PROGRAM PRG_05_Carriage
VAR
	R_TRIG_0: R_TRIG;
	R_TRIG_2: R_TRIG;
	bCarriageRt: BOOL;
	bCarriageLt: BOOL;
	lCarriageLeftLimit: LREAL;
	lCarriageRightLimit: LREAL;
	RS_CarriageCentre: RS;
	
	TOF_CarriageEN: TOF;
	R_TRIG_1: R_TRIG;
END_VAR

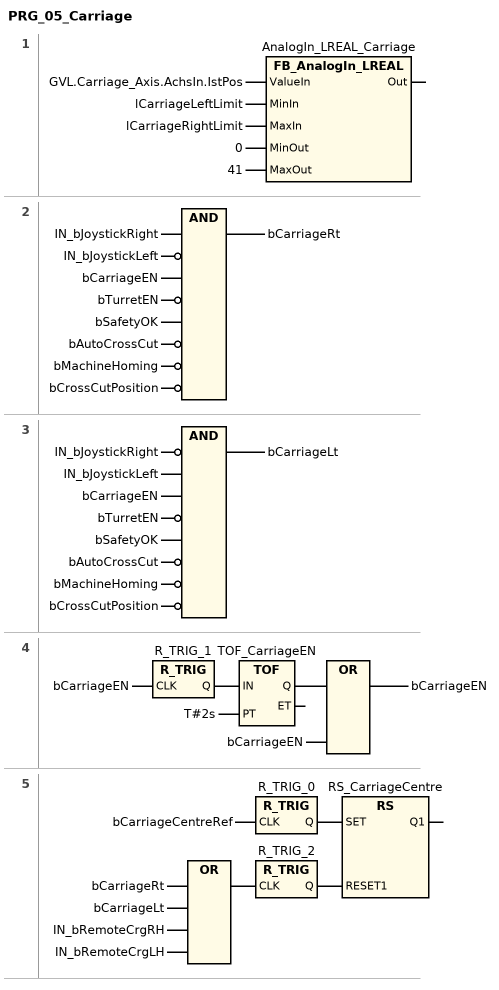
// NETWORK 1
AnalogIn_LREAL_Carriage(
    ValueIn := GVL.Carriage_Axis.AchsIn.IstPos,
    MinIn := lCarriageLeftLimit,
    MaxIn := lCarriageRightLimit,
    MinOut := 0,
    MaxOut := 41); // FB_AnalogIn_LREAL

// NETWORK 2
bCarriageRt := IN_bJoystickRight AND NOT IN_bJoystickLeft AND bCarriageEN AND NOT bTurretEN AND bSafetyOK AND NOT bAutoCrossCut AND NOT bMachineHoming AND NOT bCrossCutPosition;

// NETWORK 3
bCarriageLt := NOT IN_bJoystickRight AND IN_bJoystickLeft AND bCarriageEN AND NOT bTurretEN AND bSafetyOK AND NOT bAutoCrossCut AND NOT bMachineHoming AND NOT bCrossCutPosition;

// NETWORK 4
R_TRIG_1(CLK := bCarriageEN); // R_TRIG
TOF_CarriageEN(IN := R_TRIG_1.Q, PT := T#2s); // TOF
bCarriageEN := TOF_CarriageEN.Q OR bCarriageEN;

// NETWORK 5
R_TRIG_0(CLK := bCarriageCentreRef); // R_TRIG
R_TRIG_2(CLK := bCarriageRt OR bCarriageLt OR IN_bRemoteCrgRH OR IN_bRemoteCrgLH); // R_TRIG
RS_CarriageCentre(SET := R_TRIG_0.Q, RESET1 := R_TRIG_2.Q); // RS

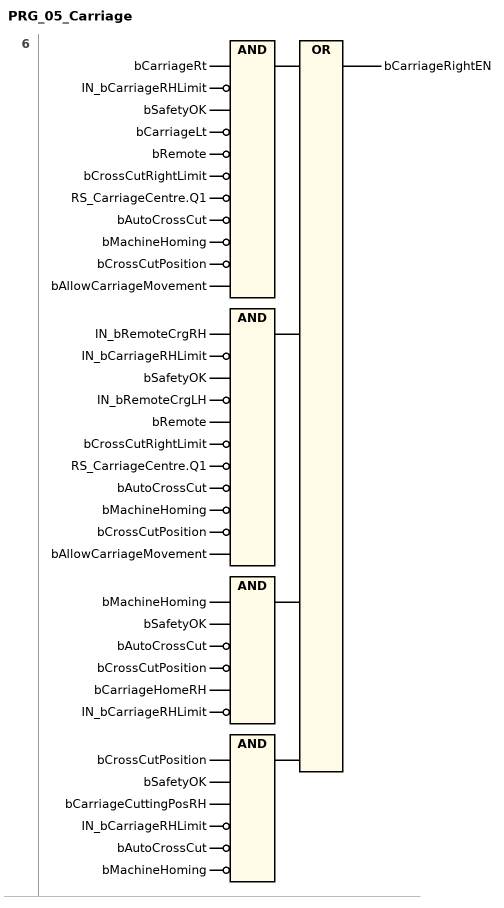
// NETWORK 6
bCarriageRightEN := bCarriageRt AND NOT IN_bCarriageRHLimit AND bSafetyOK AND NOT bCarriageLt AND NOT bRemote AND NOT bCrossCutRightLimit AND NOT RS_CarriageCentre.Q1 AND NOT bAutoCrossCut AND NOT bMachineHoming AND NOT bCrossCutPosition AND bAllowCarriageMovement OR IN_bRemoteCrgRH AND NOT IN_bCarriageRHLimit AND bSafetyOK AND NOT IN_bRemoteCrgLH AND bRemote AND NOT bCrossCutRightLimit AND NOT RS_CarriageCentre.Q1 AND NOT bAutoCrossCut AND NOT bMachineHoming AND NOT bCrossCutPosition AND bAllowCarriageMovement OR bMachineHoming AND bSafetyOK AND NOT bAutoCrossCut AND NOT bCrossCutPosition AND bCarriageHomeRH AND NOT IN_bCarriageRHLimit OR bCrossCutPosition AND bSafetyOK AND bCarriageCuttingPosRH AND NOT IN_bCarriageRHLimit AND NOT bAutoCrossCut AND NOT bMachineHoming;

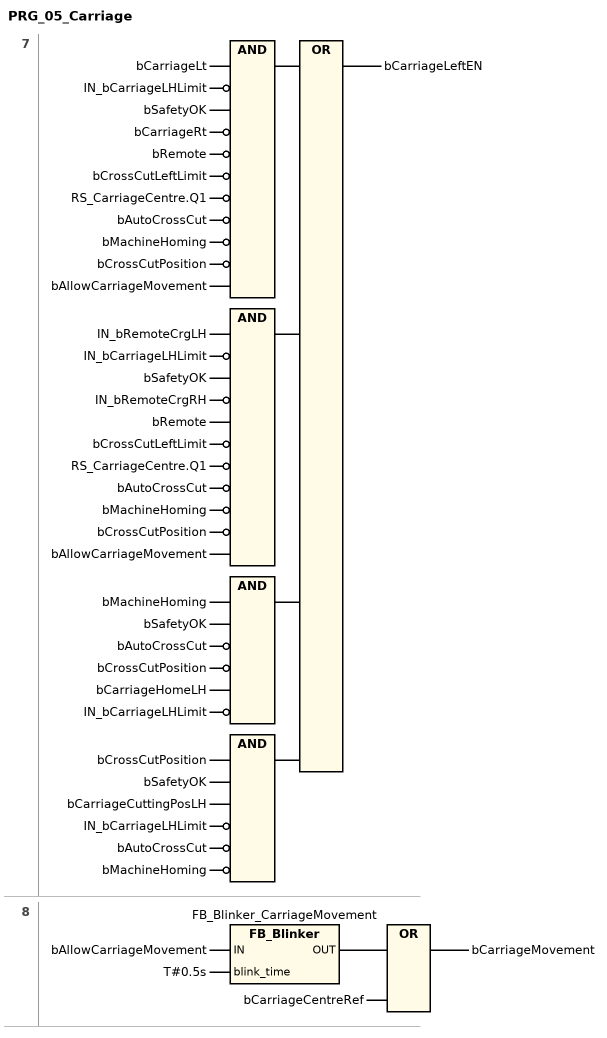
// NETWORK 7
bCarriageLeftEN := bCarriageLt AND NOT IN_bCarriageLHLimit AND bSafetyOK AND NOT bCarriageRt AND NOT bRemote AND NOT bCrossCutLeftLimit AND NOT RS_CarriageCentre.Q1 AND NOT bAutoCrossCut AND NOT bMachineHoming AND NOT bCrossCutPosition AND bAllowCarriageMovement OR IN_bRemoteCrgLH AND NOT IN_bCarriageLHLimit AND bSafetyOK AND NOT IN_bRemoteCrgRH AND bRemote AND NOT bCrossCutLeftLimit AND NOT RS_CarriageCentre.Q1 AND NOT bAutoCrossCut AND NOT bMachineHoming AND NOT bCrossCutPosition AND bAllowCarriageMovement OR bMachineHoming AND bSafetyOK AND NOT bAutoCrossCut AND NOT bCrossCutPosition AND bCarriageHomeLH AND NOT IN_bCarriageLHLimit OR bCrossCutPosition AND bSafetyOK AND bCarriageCuttingPosLH AND NOT IN_bCarriageLHLimit AND NOT bAutoCrossCut AND NOT bMachineHoming;

// NETWORK 8
FB_Blinker_CarriageMovement(IN := bAllowCarriageMovement, blink_time := T#0.5s); // FB_Blinker
bCarriageMovement := FB_Blinker_CarriageMovement.OUT OR bCarriageCentreRef;

ACTION ACT_05_1_Carriage:
lCarriageLeftLimit := 29217.032295256788 ;
lCarriageRightLimit := 30263.54710934843 ;

// Carriage centre reference trigger
IF  AnalogIn_LREAL_Carriage.Out.rScaled > 20.48 AND
	AnalogIn_LREAL_Carriage.Out.rScaled < 20.52 THEN
	bCarriageCentreRef := TRUE ;
ELSE bCarriageCentreRef := FALSE;	
END_IF

// Carriage Median
lCarriageMedian := (AnalogIn_LREAL_Carriage.MaxOut - AnalogIn_LREAL_Carriage.MinOut) / 2 ;

// Carriage slow downs approaching end limits and centre reference
IF  (AnalogIn_LREAL_Carriage.Out.rScaled <= 1 AND bCarriageLeftEN) OR
	(AnalogIn_LREAL_Carriage.Out.rScaled >= 40 AND bCarriageRightEN) OR
	(AnalogIn_LREAL_Carriage.Out.rScaled <= 21.5 AND AnalogIn_LREAL_Carriage.Out.rScaled > 20.5 AND bCarriageLeftEN) OR
	(AnalogIn_LREAL_Carriage.Out.rScaled >= 19.5 AND AnalogIn_LREAL_Carriage.Out.rScaled < 20.5 AND bCarriageRightEN) THEN
	bCarriageJogFast := FALSE ;
ELSE bCarriageJogFast := TRUE ;
END_IF
END_ACTION

END_PROGRAM

(* stored: Version 1.1.0.1, ProductVersion 3.1.4024.15
   POU PRG_05_Carriage: Id {67f21597-7dea-46f0-b94f-71ff6e827db3}, SpecialFunc None
   Action ACT_05_1_Carriage: Id {c1ab4447-ebe4-4f62-85bb-db2b3a6bc989} *)
